// TIA Portal V16 export
// export: Created 2025-05-30T16:36:17.0802048Z, ExportSetting WithDefaults, DisplayName Totally Integrated Automation Portal, DisplayVersion V16, DisplayName TIA Portal Version Control Interface, DisplayVersion V16, DisplayName TIA Portal Openness, DisplayVersion V16, DisplayName STEP 7 Professional, DisplayVersion V16, DisplayName STEP 7 Safety, DisplayVersion V16, DisplayName WinCC Advanced, DisplayVersion V16
DATA_BLOCK "IEC_Timer_0_DB_1"   // DB60
// stored: AutoNumber true, InstanceOfName TOF_SFB, OfSystemLibElement TOF, OfSystemLibVersion 1.0
"TOF_SFB"
   // VAR_INPUT
   //    IN : Bool;
   //    PT : Time;
   // END_VAR
   // VAR_OUTPUT
   //    Q : Bool;
   //    ET : Time;
   // END_VAR
   // VAR RETAIN
   //    STATE : Byte;
   //    STIME : Time;
   //    ATIME : Time;
   // END_VAR
BEGIN
END_DATA_BLOCK
